// TIA Portal V16 export
// export: Created 2021-03-15T13:24:40.4350103Z, ExportSetting WithDefaults, DisplayName Totally Integrated Automation Portal, DisplayVersion V16 Update 3, DisplayName TIA Portal Version Control Interface, DisplayVersion V16 Update 2, DisplayName TIA Portal Openness, DisplayVersion V16 Update 3, DisplayName STEP 7 Professional, DisplayVersion V16 Update 3, DisplayName STEP 7 Safety, DisplayVersion V16, DisplayName WinCC Professional, DisplayVersion V16 Update 3
TYPE "UT21000_Dy_SysSignals"
TITLE = Dynamic UDT — Sys - Global Signals
// Global Logic and Timing Signals
// stored: IsFailsafeCompliant false
   STRUCT
      revInfo { ExternalWritable := 'False'} : "UT01000_St_SysRevision";   // ▀▀▀▀ UDT CURRENT REVISION
      ___________0010_0 { ExternalAccessible := 'False'; ExternalVisible := 'False'; ExternalWritable := 'False'} : Bool;
      ___________0010_1 { ExternalAccessible := 'False'; ExternalVisible := 'False'; ExternalWritable := 'False'} : Bool;   // ▀▀▀▀ SYSTEM SIGNALS
      _False { ExternalWritable := 'False'} : Bool;   // System Logic Bit — Always FALSE
      _True { ExternalWritable := 'False'} : Bool;   // System Logic Bit — Always TRUE
      _50ms { ExternalWritable := 'False'} : Bool;   // System Timing — 50 ms Pulse Scan synchronised
      _100ms { ExternalWritable := 'False'} : Bool;   // System Timing — 100 ms Pulse Scan synchronised
      _200ms { ExternalWritable := 'False'} : Bool;   // System Timing — 200 ms Pulse Scan synchronised
      _500ms { ExternalWritable := 'False'} : Bool;   // System Timing — 500 ms Pulse Scan synchronised
      _1s { ExternalWritable := 'False'} : Bool;   // System Timing — 1 s Pulse Scan synchronised
      _2s { ExternalWritable := 'False'} : Bool;   // System Timing — 2 s Pulse Scan synchronised
      _CycleTick { ExternalWritable := 'False'} : Bool;   // System Timing — Cycle tick (active odd cycles, alternates with _CycleTock)
      _CycleTock { ExternalWritable := 'False'} : Bool;   // System Timing — Cycle tock (active even cycles, alternates with _CycleTick)
      _CycleFirst { ExternalWritable := 'False'} : Bool;   // System Timing — First cycle detected
      _100msSqW { ExternalWritable := 'False'} : Bool;   // System Timing — 100 ms Square wave Scan synchronised
      _200msSqW { ExternalWritable := 'False'} : Bool;   // System Timing — 200 ms Square wave Scan synchronised
      _500msSqW { ExternalWritable := 'False'} : Bool;   // System Timing — 500 ms Square wave Scan synchronised
      _1sSqW { ExternalWritable := 'False'} : Bool;   // System Timing — 1 s Square wave Scan synchronised
      _2sSqW { ExternalWritable := 'False'} : Bool;   // System Timing — 2 s Square wave Scan synchronised
   END_STRUCT;
   // revInfo.REV_BLOCK := 'UT21000';
   // revInfo.REV_NUMBER := '000-801';
   // revInfo.REV_DATE := '2021-02-18';
   // revInfo.REV_AUTHOR := 'M. Gledhill';
END_TYPE
